FUNCTION_BLOCK "AssemblageCel_U"
{ S7_Optimized_Access := 'TRUE' }
VERSION : 0.1
   VAR_INPUT
      Start : Bool;
      Stop : Bool;
      EStop : Bool;
   END_VAR

   VAR
      Stap : Int;
      Prev_Stap : Int;
      Lagerpers { S7_SetPoint := 'False'} : "Lagerpers_EM";
      Draaitafel : "Draaitafel_EM";
      Cobot : "Cobot_EM";
   END_VAR


BEGIN
	CASE #Stap OF
	    0:
	        #Lagerpers.StartLagerpers := FALSE;
	        IF
	            #Start THEN
	            #Stap := 1;
	        END_IF;
	    1:
	       #Cobot.I_Start_Program := TRUE;
	       IF #Cobot.Program_Completed THEN
	           #Stap := 2;
	       END_IF;
	    50: //StopState
	        IF #Start THEN
	            #Stap := #Prev_Stap;
	        END_IF;

	END_CASE;

	IF #Stop THEN
	    #Stap := 50;
	END_IF;

	#Prev_Stap := #Stap - 1;

	IF #EStop OR #Cobot.EStop_Cobot THEN
	    #Stap := 0;
	END_IF;
	#Draaitafel();
	#Cobot();
	#Lagerpers();


END_FUNCTION_BLOCK

